{attribute 'OPC.UA.DA.StructuredType' := '1'} //publikuj zmienna jako strukture
TYPE ST_AnalogSens :
STRUCT
	
	iRawValue    AT%I* : INT;	     // raw value from A/D converter PLC
	rValue  	       : REAL;       // value after conversion to real value

END_STRUCT
END_TYPE

(* stored: Version 1.1.0.1, ProductVersion 3.1.4024.15
   DUT ST_AnalogSens: Id {291d42d4-9646-45e4-a4b4-9700e8be904c} *)
